REGION Network 7: Grafcet Transport
   IF "DB_Testing".enable.Transport THEN
       "ID_PE_Transport"(i_Init := "DB_Global".transport.init OR "DB_Testing".init.Transport,   // "FB_PE_Transport"
                         i_Enable := NOT "DB_Global".general.man AND NOT "DB_Alarm".general.global,
                         i_CmdTransport := "DB_Global".transport.cmdTransport OR "DB_Testing".cmd.Transport,
                         i_CoverLoadedBit := "DB_Global".plate.currentCovers[7].loaded OR "DB_Testing".value.CoverLoaded,
                         iSenCilDown := "DB_IO".transport.iTransportSenDown,
                         iSenCilUp := "DB_IO".transport.iTransportSenUp,
                         iSenCilAtPlate := "DB_IO".transport.iTransportSenAtPlate,
                         iSenCilAtCart := "DB_IO".transport.iTransportSenAtCart,
                         io_CounterDone := "DB_Recipes".Recipes[0].Progress,
                         o_ReadyToTransport => "DB_Global".transport.sigReadyToTransport,
                         o_EmptyTransportedCoverProperties => "DB_Global".plate.currentCovers[7],
                         o_ItemPlaced => "DB_TransferPLC".ItemPlaced,
                         oVenCilDown => "DB_IO".transport.oTransportVenCilDown,
                         oVenCilToCart => "DB_IO".transport.oTransportVenCilCart,
                         oVenGripClose => "DB_IO".transport.oTransportVenGripClosed);
   END_IF;
END_REGION

REGION Network 8: ------------------------------------------------------------------------ Outputs ------------------------------------------------------------------------
END_REGION

REGION Network 9: Sturen oTransportVenCilDown_A+
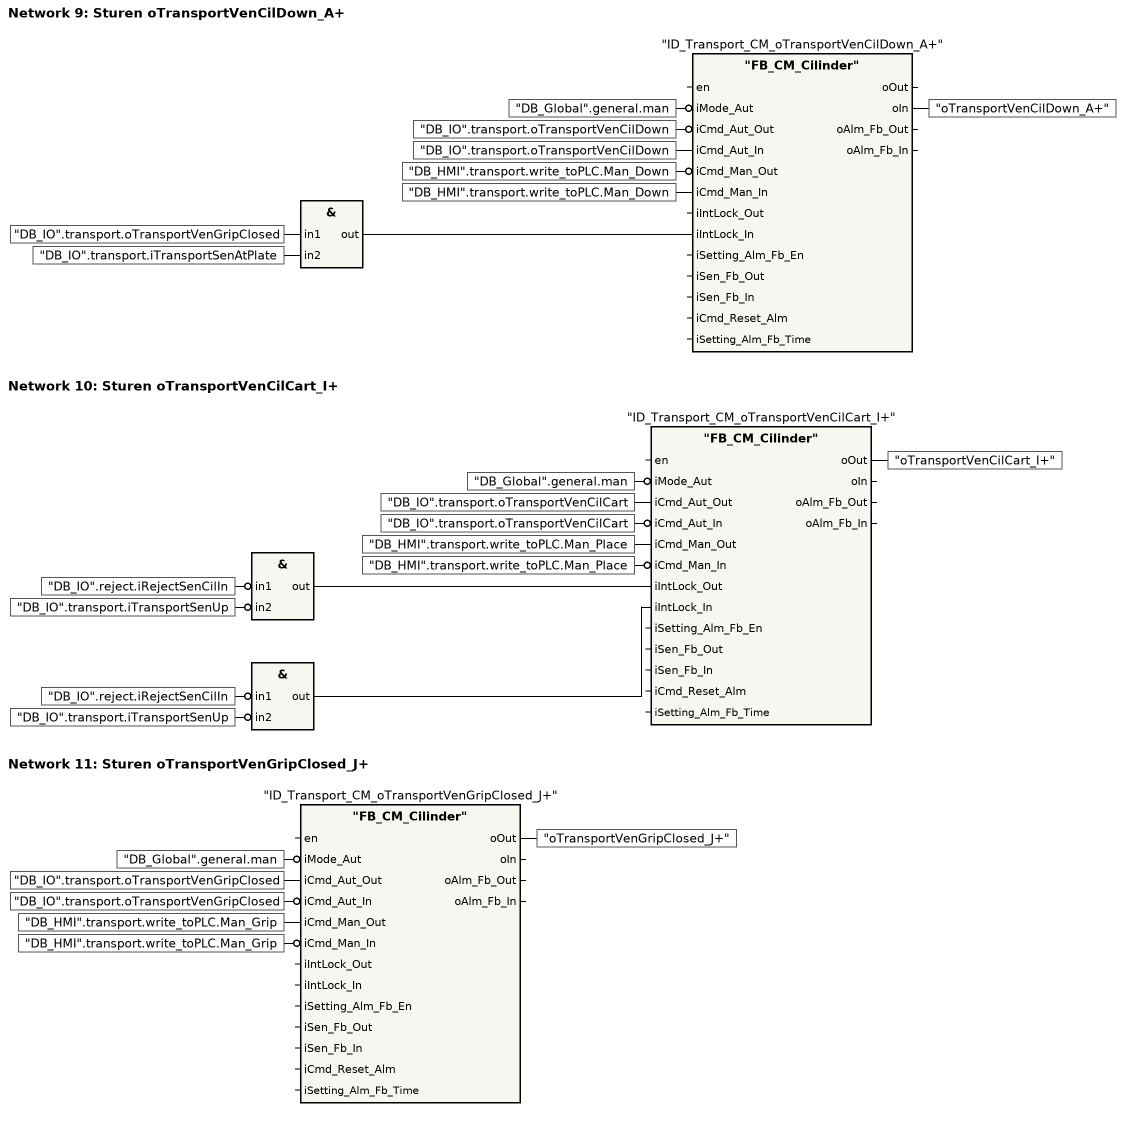
   "ID_Transport_CM_oTransportVenCilDown_A+"(iMode_Aut := NOT "DB_Global".general.man,   // "FB_CM_Cilinder"
                           iCmd_Aut_Out := NOT "DB_IO".transport.oTransportVenCilDown,
                           iCmd_Aut_In := "DB_IO".transport.oTransportVenCilDown,
                           iCmd_Man_Out := NOT "DB_HMI".transport.write_toPLC.Man_Down,
                           iCmd_Man_In := "DB_HMI".transport.write_toPLC.Man_Down,
                           iIntLock_In := "DB_IO".transport.oTransportVenGripClosed AND "DB_IO".transport.iTransportSenAtPlate,
                           oIn => "oTransportVenCilDown_A+");
END_REGION

REGION Network 10: Sturen oTransportVenCilCart_I+
   // TODO:
   // - Interlocks
   "ID_Transport_CM_oTransportVenCilCart_I+"(iMode_Aut := NOT "DB_Global".general.man,   // "FB_CM_Cilinder"
                           iCmd_Aut_Out := "DB_IO".transport.oTransportVenCilCart,
                           iCmd_Aut_In := NOT "DB_IO".transport.oTransportVenCilCart,
                           iCmd_Man_Out := "DB_HMI".transport.write_toPLC.Man_Place,
                           iCmd_Man_In := NOT "DB_HMI".transport.write_toPLC.Man_Place,
                           iIntLock_Out := NOT "DB_IO".reject.iRejectSenCilIn AND NOT "DB_IO".transport.iTransportSenUp,
                           iIntLock_In := NOT "DB_IO".reject.iRejectSenCilIn AND NOT "DB_IO".transport.iTransportSenUp,
                           oOut => "oTransportVenCilCart_I+");
END_REGION

REGION Network 11: Sturen oTransportVenGripClosed_J+
   "ID_Transport_CM_oTransportVenGripClosed_J+"(iMode_Aut := NOT "DB_Global".general.man,   // "FB_CM_Cilinder"
                           iCmd_Aut_Out := "DB_IO".transport.oTransportVenGripClosed,
                           iCmd_Aut_In := NOT "DB_IO".transport.oTransportVenGripClosed,
                           iCmd_Man_Out := "DB_HMI".transport.write_toPLC.Man_Grip,
                           iCmd_Man_In := NOT "DB_HMI".transport.write_toPLC.Man_Grip,
                           oOut => "oTransportVenGripClosed_J+");
END_REGION
END_FUNCTION

FUNCTION_BLOCK "FB_PE_Transport"
{ S7_Optimized_Access := 'TRUE' }
VERSION : 0.1
   VAR_INPUT 
      i_Init : Bool;
      i_Enable : Bool;
      i_CmdTransport : Bool;
      i_CoverLoadedBit : Bool;
      iSenCilDown : Bool;
      iSenCilUp : Bool;
      iSenCilAtPlate : Bool;
      iSenCilAtCart : Bool;
   END_VAR

   VAR_OUTPUT 
      o_ReadyToTransport : Bool;
      o_EmptyTransportedCoverProperties : "UDT_coverProperties";
      o_ItemPlaced : Bool;
      oVenCilDown : Bool;
      oVenCilToCart : Bool;
      oVenGripClose : Bool;
   END_VAR

   VAR_IN_OUT 
      io_CounterDone : Int;
   END_VAR

   VAR 
      sStep : Int;
      sInit : Bool;
      sPreviuousStep : Int;
      sTON_X1 {InstructionName := 'TON_TIME'; LibVersion := '1.0'; S7_SetPoint := 'False'} : TON_TIME;
      sTON_X2 {InstructionName := 'TON_TIME'; LibVersion := '1.0'} : TON_TIME;
      sTON_X3 {InstructionName := 'TON_TIME'; LibVersion := '1.0'} : TON_TIME;
      sTON_X4 {InstructionName := 'TON_TIME'; LibVersion := '1.0'} : TON_TIME;
      sTON_X5 {InstructionName := 'TON_TIME'; LibVersion := '1.0'} : TON_TIME;
      sTON_X6 {InstructionName := 'TON_TIME'; LibVersion := '1.0'} : TON_TIME;
      sTON_X7 {InstructionName := 'TON_TIME'; LibVersion := '1.0'} : TON_TIME;
      sTON_X8 {InstructionName := 'TON_TIME'; LibVersion := '1.0'} : TON_TIME;
      sTP_itemPlaced {InstructionName := 'TP_TIME'; LibVersion := '1.0'} : TP_TIME;
   END_VAR

   VAR CONSTANT 
      cWaitTime : Time := T#0.5s;   // With feedback
   END_VAR


BEGIN
	REGION init
	    IF #i_Init AND NOT (#sInit = #i_Init) THEN
	        #sStep := 0;
	    END_IF;
	    #sInit := #i_Init;
	END_REGION
	
	REGION enable
	    IF NOT #i_Enable THEN
	        GOTO afterGrafcetLogic;
	    END_IF;
	END_REGION
	
	REGION timers
	    
	    #sTON_X1(IN := (#sStep = 1) AND #iSenCilDown,
	             PT := #cWaitTime);
	    
	    #sTON_X2(IN := (#sStep = 2),
	             PT := #cWaitTime);
	    
	    #sTON_X3(IN := (#sStep = 3) AND #iSenCilUp,
	             PT := #cWaitTime);
	    
	    #sTON_X4(IN := (#sStep = 4) AND #iSenCilAtCart,
	             PT := #cWaitTime);
	    
	    #sTON_X5(IN := (#sStep = 5) AND #iSenCilDown,
	             PT := #cWaitTime);
	    
	    #sTON_X6(IN := (#sStep = 6),
	             PT := #cWaitTime);
	    
	    #sTON_X7(IN := (#sStep = 7) AND #iSenCilUp,
	             PT := #cWaitTime);
	    
	    #sTON_X8(IN := (#sStep = 8) AND #iSenCilAtPlate,
	             PT := #cWaitTime);
	END_REGION
	
	REGION grafcet logic
	    CASE #sStep OF
	        0:
	            IF
	                #i_CmdTransport
	                AND #i_CoverLoadedBit
	            THEN
	                #sStep := 1;
	            END_IF;
	        1:
	            IF #sTON_X1.Q THEN
	                #sStep := 2;
	            END_IF;
	        2:
	            IF #sTON_X2.Q THEN
	                #sStep := 3;
	            END_IF;
	        3:
	            IF #sTON_X3.Q THEN
	                #sStep := 4;
	            END_IF;
	        4:
	            IF #sTON_X4.Q THEN
	                #sStep := 5;
	            END_IF;
	        5:
	            IF #sTON_X5.Q THEN
	                #sStep := 6;
	            END_IF;
	        6:
	            IF #sTON_X6.Q THEN
	                #sStep := 7;
	            END_IF;
	        7:
	            IF #sTON_X7.Q THEN
	                #sStep := 8;
	            END_IF;
	        8:
	            IF #sTON_X8.Q THEN
	                #sStep := 0;
	            END_IF;
	        ELSE
	            #sStep := 0;
	    END_CASE;
	END_REGION
	
	afterGrafcetLogic: // Jump destination
	    
	REGION data management
	    
	    REGION empty loaded cover properties
	        
	        IF
	            (#sStep = 3)
	            AND NOT (#sPreviuousStep = #sStep)
	        THEN
	            // Empty picked item in array
	            #o_EmptyTransportedCoverProperties := "FC_emptyCoverProperties"();
	            // Add 1 to counter for current recipe
	            #io_CounterDone := #io_CounterDone + 1;
	        END_IF;
	    END_REGION
	    
	    REGION item placed pulse
	        
	        #sTP_itemPlaced(IN:= (#sStep = 7) AND NOT(#sPreviuousStep = #sStep),
	                        PT:= T#1.5s,
	                        Q => #o_ItemPlaced);
	        
	    END_REGION
	    
	    #sPreviuousStep := #sStep;
	    
	END_REGION
	
	REGION outputs
	    
	    #o_ReadyToTransport := #sStep = 0;
	    
	    #oVenCilDown := #sStep = 1
	                 OR #sStep = 2
	                 OR #sStep = 5
	                 OR #sStep = 6;
	    
	    #oVenCilToCart := #sStep = 4
	                   OR #sStep = 5
	                   OR #sStep = 6
	                   OR #sStep = 7;
	    
	    #oVenGripClose := #sStep = 2
	                   OR #sStep = 3
	                   OR #sStep = 4
	                   OR #sStep = 5;
	                   
	END_REGION
	
END_FUNCTION_BLOCK

FUNCTION_BLOCK "FB_CM_AnalogInput"
TITLE = FB_CM_AnalogInput AP BIB
{ S7_Optimized_Access := 'FALSE' }
VERSION : 0.1
//07/06/2023: v1 (LAJ)
   VAR_INPUT 
      iAI_Raw : Int;
      iRangeMin_EU : Real;
      iRangeMax_EU : Real;
      iSetting_Bipolar { S7_HiddenAssignment := 'Hide'} : Bool;
      iSetting_PT100 { S7_HiddenAssignment := 'Hide'} : Bool;   // if ISetting_PT100 is true, iRangeMin and iRangeMax are not used
      iSetting_CustomScale_Enable { S7_HiddenAssignment := 'Hide'} : Bool;   // if no siemens input is used, scaling is not always with 0-27648
      iSetting_CustomScale_RawMin { S7_HiddenAssignment := 'Hide'} : Int;
      iSetting_CustomScale_RawMax { S7_HiddenAssignment := 'Hide'} : Int;
   END_VAR

   VAR_OUTPUT 
      oAI_EU : Real;   // EU: engineering units
      oOutOfLimit : Bool;
   END_VAR

   VAR_TEMP 
      tScaleValueMax : Real;
      tScaleValueMin : Real;
   END_VAR


BEGIN
	//PT100
	IF #iSetting_PT100 = TRUE THEN
	    #oAI_EU := INT_TO_REAL(#iAI_Raw) / 10;
	        //alarm limit
	        IF #iAI_Raw = 32767 THEN //if PT100 not connected -> values becomes 32767
	            #oOutOfLimit := TRUE;
	        ELSE
	            #oOutOfLimit := FALSE;
	        END_IF;
	    RETURN; //ignore rest of code
	END_IF;
	
	//define tScaleValueMax en tScaleValueMin
	IF #iSetting_CustomScale_Enable = FALSE THEN //'normal' situation (siemens)
	    #tScaleValueMin := 0.0;
	    #tScaleValueMax := 27648.0;
	ELSE 
	    #tScaleValueMin := #iSetting_CustomScale_RawMin;
	    #tScaleValueMax := #iSetting_CustomScale_RawMax;
	END_IF;
	
	IF #iSetting_Bipolar = TRUE THEN
	    #tScaleValueMin := -1 * #tScaleValueMax;
	ELSE
	    #tScaleValueMin := 0.0;
	END_IF;
	
	//calculate scaled value
	#oAI_EU := #iRangeMin_EU + (((#iAI_Raw-#tScaleValueMin) / (#tScaleValueMax- #tScaleValueMin))) * (#iRangeMax_EU - #iRangeMin_EU);
	
	//out of limit
	IF #iAI_Raw > #tScaleValueMax OR #iAI_Raw < #tScaleValueMin THEN
	    #oOutOfLimit := TRUE;
	ELSE
	    #oOutOfLimit := FALSE;
	END_IF;
END_FUNCTION_BLOCK
